// TIA Portal V18 export
DATA_BLOCK "Settings"   // DB100
{ S7_Optimized_Access := 'TRUE' }
// stored: AutoNumber false, MemoryReserve 100
   VAR RETAIN
      ActTorqAlpha { S7_SetPoint := 'True'} : Real := 0.0;   // Low Pass Filter, Alpha be >= 0 and < 1. 0 No filterting.
      AlarmDebounce { S7_SetPoint := 'True'} : Time := T#500MS;   // Time an alarm must be present before setting
      MUTorqAutoSet1per { S7_SetPoint := 'True'} : Real := 65.0;   // Perfent of MU a torq low Set point to allow full speed ramp
      MUTorqAutoSet2per { S7_SetPoint := 'True'} : Real := 90.0;   // Percent of MU Torq high setpoint to say complete
      MUAutoHoldTime { S7_SetPoint := 'True'} : Time := T#2S_150MS;   // Time System will hold max torq before ramping down
      MUAutoSlewLow { S7_SetPoint := 'True'} : Real := 150.0;   // Slew rate for Auto make up rising in low torque. mA/Sec
      MUAutoSlewMid { S7_SetPoint := 'True'} : Real := 25.0;   // Slew rate for Auto make up rising in mid torq. mA/Sec
      AuxFlowMinGPM { S7_SetPoint := 'True'} : Real := 5.0;   // Min Value of flow transducer
      AuxFlowMaxGPM { S7_SetPoint := 'True'} : Real := 25.0;   // MAx Value of flow transducer
      AuxFlowAlpha { S7_SetPoint := 'True'} : Real := 0.0;   // Low Pass Filter, Alpha be >= 0 and < 1. 0 No filterting.
      BOFlowSlewRise { S7_SetPoint := 'True'} : Real := 500.0;   // Rising Slew Rate mA/sec on Flow Output
      BOFlowSlewFall { S7_SetPoint := 'True'} : Real := 80.0;   // Falling Slew Rate mA/sec on Flow Output
      BOSpinFactor { S7_SetPoint := 'True'} : Real := 1.25;   // BO Flow will be set to MU Spin Percent times this factor to break connection. before slowing back down to Spin Speed
      BOShiftRPM { S7_SetPoint := 'True'} : Real := 4.0;   // In BO above this speed, system will switch from BO Speed setting to Spin setting
      BypassTime { S7_SetPoint := 'True'} : Time := T#2S;   // Time for Bypass to finish running
      BypassFlowPer { S7_SetPoint := 'True'} : Real := 50.0;   // Output to flow in percent valve in Bypass mode
      BypassTorqFtlbs { S7_SetPoint := 'True'} : Real := 12000.0;   // Output to torqur valve in Bypass mode. Actual Value TBD
      CATEngPPR { S7_SetPoint := 'True'} : Int := 113;   // CAT Engine PPR.
      CATMinRPM { S7_SetPoint := 'True'} : Real := 1200.0;   // Minimum running RPM of CAT. Used to trigger Enginer fault
      CATFaultTime { S7_SetPoint := 'True'} : Time := T#15S;   // Time for CAT to get up to speed before fault
      ChargeFlowMinGPM { S7_SetPoint := 'True'} : Real := 5.0;   // Min Value of flow transducer
      ChargeFlowMaxGPM { S7_SetPoint := 'True'} : Real := 1000.0;   // MAx Value of flow transducer
      ChargeFlowAlpha { S7_SetPoint := 'True'} : Real := 0.0;   // Low Pass Filter, Alpha be >= 0 and < 1. 0 No filterting.
      ChargePress1Min { S7_SetPoint := 'True'} : Real := 0.0;   // Min value of transducer range
      ChargePress1Max { S7_SetPoint := 'True'} : Real := 6000.0;   // Max Value of transducer range
      ChargePress1Alpha { S7_SetPoint := 'True'} : Real := 0.0;   // Low Pass Filter, Alpha be >= 0 and < 1. 0 No filterting.
      ChargePress2Min { S7_SetPoint := 'True'} : Real := 0.0;   // Min value of transducer range
      ChargePress2Max { S7_SetPoint := 'True'} : Real := 6000.0;   // Max Value of transducer range
      ChargePress2Alpha { S7_SetPoint := 'True'} : Real := -7111.111;   // Low Pass Filter, Alpha be >= 0 and < 1. 0 No filterting.
      ChargeFaultMinPress { S7_SetPoint := 'True'} : Real := 200.0;   // Min charge pressure before fault shown
      ChargeFaultMaxPress { S7_SetPoint := 'True'} : Real := 1000.0;   // Max Charge pressure before fautl
      CLTempMinC { S7_SetPoint := 'True'} : Real := 0.0;   // Min value of Closed loop Temp transducer
      CLTempMaxC { S7_SetPoint := 'True'} : Real := 204.0;   // Max value of Closed loop Temp transducer
      CLTempMinF { S7_SetPoint := 'True'} : Real := 0.0;
      CLTempMaxF { S7_SetPoint := 'True'} : Real := 400.0;
      CLTempAlpha { S7_SetPoint := 'True'} : Real := 0.0;   // Low Pass Filter, Alpha be >= 0 and < 1. 0 No filterting.
   END_VAR
   VAR
      CLHiTempAlarmF : Real := 158.0;
   END_VAR
   VAR RETAIN
      CLHiTempAlarm { S7_SetPoint := 'True'} : Real := 70.0;   // Closed loop temp in C where alarm comes on. Value for Mobil SCH S26 - Hydrex MV60 - 64
   END_VAR
   VAR
      CLHiTempRPMF : Real := 161.6;
   END_VAR
   VAR RETAIN
      ClHiTempRPM { S7_SetPoint := 'True'} : Real := 72.0;   // Closed loop temp in c where RPM is reduced Value for Mobil SCH S26 - Hydrex MV60 - 66
   END_VAR
   VAR
      ClHiTempShutdownF : Real := 165.2;
   END_VAR
   VAR RETAIN
      ClHiTempShutdown { S7_SetPoint := 'True'} : Real := 74.0;   // Closed loop temp in C where TD shutsdown Value for Mobil SCH S26 - Hydrex MV60 - 68
   END_VAR
   VAR
      ClHiTempBypassF : Real := 161.6;
   END_VAR
   VAR RETAIN
      ClHiTempBypass { S7_SetPoint := 'True'} : Real := 72.0;   // Closed loop Temp in C where Bypass stopped Value for Mobil SCH S26 - Hydrex MV60 - 66
      ClHiTempRPMmA { S7_SetPoint := 'True'} : Real := 410.0;   // The max mA output in high temp reduced RPM mode
      CoolingFanTempC { S7_SetPoint := 'True'} : Real := 65.0;   // Temperature at which point cooling fan will turn on
      CoolingFanTimeOn { S7_SetPoint := 'True'} : Time := T#30S;   // The time the cooling fan will stay on for after temp below setpoint
      DrillTorqPotAlpha { S7_SetPoint := 'True'} : Real := 0.0;   // Low Pass Filter, Alpha be >= 0 and < 1. 0 No filterting.
      DrillThrottleAlpha { S7_SetPoint := 'True'} : Real := 0.0;   // Low Pass Filter, Alpha be >= 0 and < 1. 0 No filterting.
      DrillTorqLimLowPer { S7_SetPoint := 'True'} : Real := 80.0;   // Percent of Drill a torq Low Set point to allow before destroke flow for torq limit
      DrillTorqLimHighPer { S7_SetPoint := 'True'} : Real := 97.0;   // Percent of Drill a torq High Set point before destroke flow for torq limit
      DrillTorqLimTime { S7_SetPoint := 'True'} : Time := T#50MS;   // Debounce time that torq can be above low limit before limiting flow.
      DrillTorqLimSlewRise { S7_SetPoint := 'True'} : Real := 5.0;   // Rising Slew Rate mA/sec on Torq output not in Auto Mode
      DrillTorqLimSlewFall { S7_SetPoint := 'True'} : Real := 20.0;   // Falling Slew Rate mA/sec on Torq output not in Auto Mode
      FlushFlowFaultTime { S7_SetPoint := 'True'} : Time := T#10S;   // Time with flow while aux pump is running before fault
      HeartbeatTimeout { S7_SetPoint := 'True'} : Time := T#3S;   // Time heartbeat signal can remain unchanged before IO is dropped from remote console.
      HotOilFlowMinGPM { S7_SetPoint := 'True'} : Real := 5.0;   // Min Value of flow transducer
      HotOilFlowMaxGPM { S7_SetPoint := 'True'} : Real := 1000.0;   // MAx Value of flow transducer
      HotOilFlowAlpha { S7_SetPoint := 'True'} : Real := 0.0;   // Low Pass Filter, Alpha be >= 0 and < 1. 0 No filterting.
      HornOnTime { S7_SetPoint := 'True'} : Time := T#1S_500MS;   // Time horn output is on when horn requested
      HornSilenceTime { S7_SetPoint := 'True'} : Time := T#30S;   // Time horn will turn off if high temp shutdown
      HSLTShiftTime { S7_SetPoint := 'True'} : Time := T#2S;   // Time to allow system to shift before outputting to pump
      LampTestTime { S7_SetPoint := 'True'} : Time := T#2S;   // Time lamps will be on during lamp test
      LamptTestHornTime : Time := T#2S;   // Time horn will be on during lamp test
      LSHTShiftTime { S7_SetPoint := 'True'} : Time := T#4S;   // Time to allow system to shift before outputting to pump
      LubeFlowFaultTime { S7_SetPoint := 'True'} : Time := T#10S;   // Time After aux pump runnign before flow to be seen or alarm
      M1CurrentMin { S7_SetPoint := 'True'} : Real := 0.0;   // Min value of M1 Current Input- TBD actual values
      M1CurrentMax { S7_SetPoint := 'True'} : Real := 100.0;   // Max value of M1 Current Input- TBD actual values
      M1CurrentAlpha { S7_SetPoint := 'True'} : Real := 0.0;   // Low Pass Filter, Alpha be >= 0 and < 1. 0 No filterting.
      M2CurrentMin { S7_SetPoint := 'True'} : Real := 0.0;   // Min value of M2 Current Input- TBD actual values
      M2CurrentMax { S7_SetPoint := 'True'} : Real := 100.0;   // Max value of M2 Current Input - TBD actual values
      M2CurrentAlpha { S7_SetPoint := 'True'} : Real := 0.0;   // Low Pass Filter, Alpha be >= 0 and < 1. 0 No filterting.
      MotorFaultTime { S7_SetPoint := 'True'} : Time := T#15S;   // Time before signalling a motor fault if not started after start signal sent
      MUDoneTHper { S7_SetPoint := 'True'} : Real := 60.0;   // Torque threshold percent to determne mu done
      MUSpinAdjInc { S7_SetPoint := 'True'} : Real := 5.0;   // Increment in which the MU Spin value will adjust when requested
      MUSpinMaxSpeedPer { S7_SetPoint := 'True'} : Real := 80.0;   // The MU Spin max setting to limit user adjustment
      MUSpinTorqFtlbs { S7_SetPoint := 'True'} : Real := 2000.0;   // MU Spin torq settings. If Actual torq above this value spin complete
      MUTorqSlewRise { S7_SetPoint := 'True'} : Real := 45.0;   // Rising Slew Rate mA/sec on Torq output not in Auto Mode
      MUTorqSlewFall { S7_SetPoint := 'True'} : Real := 150.0;   // Falling Slew Rate mA/sec on Torq output not in Auto Mode
      MUFlowSlewRise { S7_SetPoint := 'True'} : Real := 25.0;   // Rising Slew Rate mA/sec on Flow Output
      MUFlowSlewFall { S7_SetPoint := 'True'} : Real := 150.0;   // Falling Slew Rate mA/sec on Flow Output
      MUFlowMinmA { S7_SetPoint := 'True'} : Real := 150.0;   // Min mA Output to Flow Pump in MU Torq
      MUFlowMaxmA { S7_SetPoint := 'True'} : Real := 800.0;   // Max mA Output to Flow Pump in MU Torq
      MUTorqPotAlpha { S7_SetPoint := 'True'} : Real := 0.0;   // Low Pass Filter, Alpha be >= 0 and < 1. 0 No filterting.
      OscMaxSpeedRPM { S7_SetPoint := 'True'} : Real := 30.0;   // Maximum rotary speed setpoint allowed for Oscialltor operation.
      OscMaxTorqFtLbs { S7_SetPoint := 'True'} : Real := 20000.0;   // Maximum torq setpoint allowed for Oscialltor operation.
      OscTorqLimLowPer { S7_SetPoint := 'True'} : Real := 90.0;   // Percent of Osc torq Low Set point to allow before destroke flow for torq limit
      OscTorqLimHighPer { S7_SetPoint := 'True'} : Real := 97.0;   // Percent of Osc torq High Set point before destroke flow for torq limit
      OscTorqLimTime { S7_SetPoint := 'True'} : Time := T#1MS;   // Debounce time that torq can be above low limit before limiting flow.
      PotZero { S7_SetPoint := 'True'} : Real := 5.0;   // Any percentage below this will be considered a zero input from the throttle.
      PumpOutMinmA { S7_SetPoint := 'True'} : Real := 200.0;   // Minimum mA setting to valve
      PumpOutMaxmA { S7_SetPoint := 'True'} : Real := 700.0;   // MaximummA setting to valve
      RotEncPPR { S7_SetPoint := 'True'} : Int := 22;   // Rotatry Encoder Counts per revolution
      RotStoppedTime { S7_SetPoint := 'True'} : Time := T#2S;   // Time without an encoder count before declaring stopped.
      SpeedLimLowRPM { S7_SetPoint := 'True'} : Real := 183.0;   // Speed limiter lower threshold
      SpeedLimHighRPM { S7_SetPoint := 'True'} : Real := 190.0;   // Speed limiter upper threshold
      SpeedLimSlewRise { S7_SetPoint := 'True'} : Real := 10.0;   // Rising Slew Rate mA/sec on Flow Output
      SpeedLimSlewFall { S7_SetPoint := 'True'} : Real := 10.0;   // Falling Slew Rate mA/sec on Flow Output
      SpinSpeedPer { S7_SetPoint := 'True'} : Real := 25.0;   // TheSpin speed setting in percent. User adjustable with Link Tilt. Value used for BO Spin also
      TDFwdPressMin { S7_SetPoint := 'True'} : Real := 0.0;   // Min value of TD Fwd Press transducer
      TDFwdPressMax { S7_SetPoint := 'True'} : Real := 5800.0;   // Max value of TD Fwd Press transducer
      TDFwdPressAlpha { S7_SetPoint := 'True'} : Real := 0.0;   // Low Pass Filter, Alpha be >= 0 and < 1. 0 No filterting.
      TDRevPressMax { S7_SetPoint := 'True'} : Real := 5800.0;   // Max value of TD Rev Press transducer
      TDRevPressMin { S7_SetPoint := 'True'} : Real := 0.0;   // Min value of TD Rev Press transducer
      TDRevPressAlpha { S7_SetPoint := 'True'} : Real := 0.0;   // Low Pass Filter, Alpha be >= 0 and < 1. 0 No filterting.
      TorqEFactorLow { S7_SetPoint := 'True'} : Real := 0.97;   // 0-1. Efficiency of Torque reading when below 5 RPM
      TorqEFactorHigh { S7_SetPoint := 'True'} : Real := 0.97;   // 0-1. Efficiency of Torque reading when below 5 RPM
      TorqInHSLT { S7_SetPoint := 'True'} : Real := 3.56;   // ft-lbs /psi in High speed low torque.
      TorqInLSHT { S7_SetPoint := 'True'} : Real := 7.119;   // ft-lbs / psi in low speed high torque.
      TorqPotMaxFtLbs { S7_SetPoint := 'True'} : Real := 30000.0;   // Max value in ft-lbs that the input pot should read(Actual value TBD)
      TorqOutExtraPSI { S7_SetPoint := 'True'} : Real := 51.60006;   // Extra PSI value added to torque output to overcome charge pressure
      TorqOutMinmA { S7_SetPoint := 'True'} : Real := 100.0;   // Minimum mA setting to valve
      TorqOutMaxmA { S7_SetPoint := 'True'} : Real := 800.0;   // MaximummA setting to valve
      TorqOutMinPSI { S7_SetPoint := 'True'} : Real := 0.0;   // Minimum PSI setting on Torq valve
      TorqOutMaxPSI { S7_SetPoint := 'True'} : Real := 5075.0;   // Maximum PSI setting on Torq Valve
      TorqOutHSLT { S7_SetPoint := 'True'} : Real := 3.56;   // ft-lbs /psi at output vavle in High speed low torque. Current values are same as Feedback actual value TBD
      TorqOutLSHT { S7_SetPoint := 'True'} : Real := 7.119;   // ft-lbs / psi output vavle in low speed high torque.Current values are same as Feedback actual value TBD
      TorqSetFactor { S7_SetPoint := 'True'} : Real := 1.0;   // Torq setpoint factor to increase the setpoint to ensure desired torq is reached. Torq limiting will be controlled via flow.
   END_VAR
BEGIN
END_DATA_BLOCK
